// TIA Portal V17 export
// export: Created 2022-07-16T16:56:06.8106579Z, ExportSetting WithDefaults, DisplayName Totally Integrated Automation Portal, DisplayVersion V17, DisplayName TIA Portal Openness, DisplayVersion V17, DisplayName TIA Portal Version Control Interface, DisplayVersion V17, DisplayName TIA Portal Test Suite Advanced, DisplayVersion V17, DisplayName STEP 7 Professional, DisplayVersion V17, DisplayName STEP 7 Safety, DisplayVersion V17, DisplayName WinCC Professional, DisplayVersion V17
ORGANIZATION_BLOCK "Main"   // OB1, LAD, ProgramCycle
TITLE = "Main Program Sweep (Cycle)"
{ S7_Optimized_Access := 'TRUE' }
VERSION : 0.1
// stored: AutoNumber true, IsIECCheckEnabled false, SetENOAutomatically false
   VAR_INPUT
      Initial_Call : Bool;   // Initial call of this OB
      Remanence : Bool;   // =True, if remanent data are available
   END_VAR
BEGIN

REGION Network 1
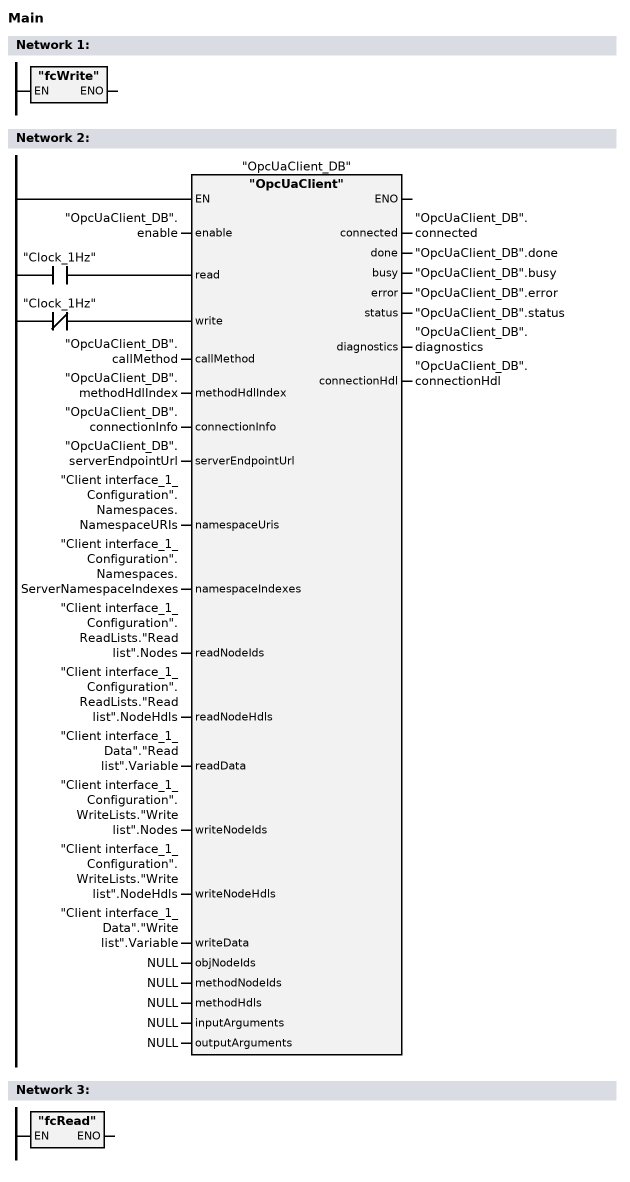
   RUNG wire#powerrail
      "fcWrite"()
   END_RUNG
   // the same network as SCL:
   "fcWrite"();
END_REGION

REGION Network 2
   RUNG wire#powerrail
      "OpcUaClient_DB"(read := wire#w1, write := wire#w2, enable := "OpcUaClient_DB".enable, callMethod := "OpcUaClient_DB".callMethod, methodHdlIndex := "OpcUaClient_DB".methodHdlIndex, connectionInfo := "OpcUaClient_DB".connectionInfo, serverEndpointUrl := "OpcUaClient_DB".serverEndpointUrl, namespaceUris := "Client interface_1_Configuration".Namespaces.NamespaceURIs, namespaceIndexes := "Client interface_1_Configuration".Namespaces.ServerNamespaceIndexes, readNodeIds := "Client interface_1_Configuration".ReadLists."Read list".Nodes, readNodeHdls := "Client interface_1_Configuration".ReadLists."Read list".NodeHdls, readData := "Client interface_1_Data"."Read list".Variable, writeNodeIds := "Client interface_1_Configuration".WriteLists."Write list".Nodes, writeNodeHdls := "Client interface_1_Configuration".WriteLists."Write list".NodeHdls, writeData := "Client interface_1_Data"."Write list".Variable, objNodeIds := NULL, methodNodeIds := NULL, methodHdls := NULL, inputArguments := NULL, outputArguments := NULL, connected => "OpcUaClient_DB".connected, done => "OpcUaClient_DB".done, busy => "OpcUaClient_DB".busy, error => "OpcUaClient_DB".error, status => "OpcUaClient_DB".status, diagnostics => "OpcUaClient_DB".diagnostics, connectionHdl => "OpcUaClient_DB".connectionHdl)
   END_RUNG
   RUNG wire#powerrail
      Contact( "Clock_1Hz" )
   END_RUNG wire#w1
   RUNG wire#powerrail
      I_Contact( "Clock_1Hz" )
   END_RUNG wire#w2
   // the same network as SCL:
   "OpcUaClient_DB"(enable := "OpcUaClient_DB".enable,   // "OpcUaClient"
                    read := "Clock_1Hz",
                    write := NOT "Clock_1Hz",
                    callMethod := "OpcUaClient_DB".callMethod,
                    methodHdlIndex := "OpcUaClient_DB".methodHdlIndex,
                    connectionInfo := "OpcUaClient_DB".connectionInfo,
                    serverEndpointUrl := "OpcUaClient_DB".serverEndpointUrl,
                    namespaceUris := "Client interface_1_Configuration".Namespaces.NamespaceURIs,
                    namespaceIndexes := "Client interface_1_Configuration".Namespaces.ServerNamespaceIndexes,
                    readNodeIds := "Client interface_1_Configuration".ReadLists."Read list".Nodes,
                    readNodeHdls := "Client interface_1_Configuration".ReadLists."Read list".NodeHdls,
                    readData := "Client interface_1_Data"."Read list".Variable,
                    writeNodeIds := "Client interface_1_Configuration".WriteLists."Write list".Nodes,
                    writeNodeHdls := "Client interface_1_Configuration".WriteLists."Write list".NodeHdls,
                    writeData := "Client interface_1_Data"."Write list".Variable,
                    objNodeIds := NULL,
                    methodNodeIds := NULL,
                    methodHdls := NULL,
                    inputArguments := NULL,
                    outputArguments := NULL,
                    connected => "OpcUaClient_DB".connected,
                    done => "OpcUaClient_DB".done,
                    busy => "OpcUaClient_DB".busy,
                    error => "OpcUaClient_DB".error,
                    status => "OpcUaClient_DB".status,
                    diagnostics => "OpcUaClient_DB".diagnostics,
                    connectionHdl => "OpcUaClient_DB".connectionHdl);
END_REGION

REGION Network 3
   RUNG wire#powerrail
      "fcRead"()
   END_RUNG
   // the same network as SCL:
   "fcRead"();
END_REGION
END_ORGANIZATION_BLOCK
